Yaskawa INFORM job: P_YR.JBI

/JOB
//NAME P_YR
///FOLDERNAME INNE
//POS
///NPOS 7,7,7,0,0,0
///TOOL 0
///POSTYPE PULSE
///PULSE
C00000=31431,-29828,24524,8917,77861,9226
C00001=30003,3333,49147,8491,79862,8933
C00002=18157,42086,87625,5262,76992,5257
C00003=-10967,57528,106023,-3217,73935,-3090
C00004=-23075,23798,68147,-6582,79268,-6819
C00005=-30125,-5252,42026,-8503,79831,-8969
C00006=-26716,-38630,19277,-7644,77005,-7765
BC00000=103636,1063121,678621
BC00001=103636,1063121,678621
BC00002=103636,1063121,678621
BC00003=103636,1063121,678621
BC00004=103636,1063121,678621
BC00005=103636,1063121,678621
BC00006=103636,1063121,678621
EC00000=0,0
EC00001=0,239555
EC00002=0,501510
EC00003=0,982190
EC00004=0,1204752
EC00005=0,1402700
EC00006=0,1659361
//INST
///DATE 2023/10/04 15:13
///ATTR SC,RW
///GROUP1 RB1,BS1
///GROUP2 ST1
NOP
MOVJ C00000 BC00000 VJ=0.78  +MOVJ EC00000 VJ=0.78
MOVJ C00001 BC00001 VJ=0.78  +MOVJ EC00001 VJ=0.78
MOVJ C00002 BC00002 VJ=0.78  +MOVJ EC00002 VJ=0.78
MOVJ C00003 BC00003 VJ=0.78  +MOVJ EC00003 VJ=0.78
MOVJ C00004 BC00004 VJ=0.78  +MOVJ EC00004 VJ=0.78
MOVJ C00005 BC00005 VJ=0.78  +MOVJ EC00005 VJ=0.78
MOVJ C00006 BC00006 VJ=0.78  +MOVJ EC00006 VJ=0.78
END
